FUNCTION_BLOCK Test_TStreamAdd_DetectsUnexpectedType EXTENDS T_UnitTestBase
VAR
    Stream : T_Stream(StreamLength := 2);
END_VAR



Stream.Init(2);

Stream.Add_INT(1234);
    
Stream.Seek(0);

// check that reading the wrong type returns zero
Assertion.AssertEquals_UINT(
    Expected := 0,
    Actual := Stream.Read_UINT(),
    VariableName := 'Stream.Read_UINT()');
    
// check the read pointer is restored...
Assertion.AssertEquals_UDINT(
    Expected := 0,
    Actual := Stream.Position,
    VariableName := 'Stream.Position');
    
    
TestFinished();

END_FUNCTION_BLOCK

(* stored: Version 1.1.0.1, ProductVersion 3.1.4024.6
   POU Test_TStreamAdd_DetectsUnexpectedType: Id {1360d495-e9de-41ec-9150-13951a2d63ad}, SpecialFunc None *)
